// SIMATIC S7-200 project (STEP 7-Micro/WIN), CPU 222 REL 02.01

SYMBOL_TABLE USER1
AUTO             I0.0     // SELEZIONE MODO DI FUNZIONAMENTO AUTOMATICO
SEMI_AUTO        I0.1     // SELEZIONE MODO DI FUNZIONAMENTO SEMI-AUTOMATICO
MANU             I0.2     // SELEZIONE MODO DI FUNZIONAMENTO MANUALE
B7               I0.3     // TRASCINATORE
B8               I0.4     // TRASCINATORE
E1               I0.5     // ESPULSORE 1 MANUALE
E2               I0.6     // ESPULSORE 2 MANUALE
B1               I0.7     // RELE' FOTOELETTRICO
B2               I1.0     // RELE' FOTOELETTRICO
B3               I1.1     // RELE' FOTOELETTRICO
B4               I1.2     // RELE' FOTOELETTRICO BOX1
B5               I1.3     // RELE' FOTOELETTRICO BOX2
B6               I1.4     // RELE' FOTOELETTRICO FINE LINEA
MANU_RICH_TR     I1.5     // COMANDO MANUALE RICHIESTA TRONCHI
CORTO            M0.0     // RILEVATO TRONCO CORTO
MEDIO            M0.1     // RILEVATO TRONCO MEDIO
LUNGO            M0.2     // RILEVATO TRONCO LUNGO
MEM_T_EVAQ       M1.0     // MEMORIA PER CONSENTIRE L'USCITA DEL TRONCO A FINE LINEA
MEM_T_DEP_BOX2   M1.1     // MEMORIA MEMORIA PER CONSENTIRE IL DEPOSITO DEL TRONCO NEL BOX 2
MEM_T_DEP_BOX1   M1.2     // MEMORIA MEMORIA PER CONSENTIRE IL DEPOSITO DEL TRONCO NEL BOX 1
ESP1             Q0.0     // MOVIMENTO ESPULSORE 1
ESP2             Q0.1     // MOVIMENTO ESPULSORE 2
AUT_RICH_TR      Q0.2     // RICHIESTA TRONCHI
T_ATT_FINE       T39      // TEMPO ATTESA USCTA SU FINE LINEA
T_ATT_BOX_2      T40      // TEMPO ATTESA DEPOSITO SU BOX 2
T_ATT_BOX_1      T41      // TEMPO ATTESA DEPOSITO SU BOX  1
END_SYMBOL_TABLE

ORGANIZATION_BLOCK MAIN:OB1
TITLE=DP208 SELEZIONE LUNGHEZZE
BEGIN
Network 1 // COMMUTA SUL FUNZIONAMENTO MANUALE
LD     MANU:I0.2
CALL   MANUALE:SBR3
Network 2 // COMMUTA SUL FUNZIONAMENTO SEMI AUTOMATICO
LD     SEMI_AUTO:I0.1
CALL   SEMIAUTOMATICO:SBR0
Network 3 // COMMUTA SUL FUNZIONAMENTO AUTOMATICO
LD     AUTO:I0.0
CALL   AUTOMATICO:SBR1
Network 4 // ESEGUE LA SELEZIONE DEL FORMATO 
LD     SM0.0
CALL   SELEZIONE:SBR2
END_ORGANIZATION_BLOCK

SUBROUTINE_BLOCK SEMIAUTOMATICO:SBR0
TITLE=FUNZIONAMENTO SEMI-AUTOMATICO
BEGIN
Network 1 // RICHIAMO TRONCO
// RICHIAMO TRONCHI:
// - RICHIESTA MANUALE DA PULSANTE
// - RICHIESTA AUTOMATICA DOPO ATTESA TRANSITO COMPLETO DEL TRONCO PRECEDENTE
LD     T_ATT_FINE:T39
O      T_ATT_BOX_2:T40
O      T_ATT_BOX_1:T41
O      MANU_RICH_TR:I1.5
=      AUT_RICH_TR:Q0.2
=      Q0.3
Network 2 // USCITA TRONCO LUNGO
// RITARDO INTENZIONALE PRIMA DI RICHIAMARE IL TRONCO SUCCESSIVO
// PER CONSENTIRE L'USCITA DEL TRONCO LUNGO
LD     B6:I1.4
ED
O      MEM_T_EVAQ:M1.0
LPS
AW<=   T_ATT_FINE:T39, 60
=      MEM_T_EVAQ:M1.0
LPP
TON    T_ATT_FINE:T39, +50
Network 3 // USCITA  TRONCO MEDIO
// RITARDO INTENZIONALE PRIMA DI RICHIAMARE IL TRONCO SUCCESSIVO
// PER CONSENTIRE IL DEPOSITO DEL TRONCO MEDIO NEL BOX 2
LD     B5:I1.3
ED
O      MEM_T_DEP_BOX2:M1.1
LPS
AW<=   T_ATT_BOX_2:T40, 30
=      MEM_T_DEP_BOX2:M1.1
LPP
TON    T_ATT_BOX_2:T40, 20
Network 4 // USCITA TRONCO CORTO
// RITARDO INTENZIONALE PRIMA DI RICHIAMARE IL TRONCO SUCCESSIVO
// PER CONSENTIRE IL DEPOSITO DEL TRONCO CORTO NEL BOX 1
LD     B4:I1.2
ED
O      MEM_T_DEP_BOX1:M1.2
LPS
AW<=   T_ATT_BOX_1:T41, 30
=      MEM_T_DEP_BOX1:M1.2
LPP
TON    T_ATT_BOX_1:T41, 20
Network 5 // COMANDO ESPULSORE 1
// SE IL TRONCO E' DEL FORMATO CORTO E VIENE COMANDATO L'ESPULSORE E1
// IL TRONCO VIENE DEPOSITATO NEL BOX 1
LD     CORTO:M0.0
A      E1:I0.5
=      ESP1:Q0.0
Network 6 // COMANDO ESPULSORE 2
// SE IL TRONCO E' DEL FORMATO MEDIO E VIENE COMANDATO L'ESPULSORE E2
// IL TRONCO VIENE DEPOSITATO NEL BOX 2
LD     MEDIO:M0.1
A      E2:I0.6
=      ESP2:Q0.1
Network 13 // Titolo del segmento
// Commento del segmento
END_SUBROUTINE_BLOCK

SUBROUTINE_BLOCK AUTOMATICO:SBR1
TITLE=FUNZIONAMENTO AUTOMATICO
BEGIN
Network 1 // RICHIAMO TRONCO
// RICHIAMO TRONCHI:
// - RICHIESTA MANUALE DA PULSANTE
// - RICHIESTA AUTOMATICA DOPO ATTESA TRANSITO COMPLETO DEL TRONCO PRECEDENTE
LD     T_ATT_FINE:T39
O      T_ATT_BOX_2:T40
O      T_ATT_BOX_1:T41
O      MANU_RICH_TR:I1.5
=      AUT_RICH_TR:Q0.2
=      Q0.3
Network 2 // USCITA TRONCO LUNGO
// RITARDO INTENZIONALE PRIMA DI RICHIAMARE IL TRONCO SUCCESSIVO
// PER CONSENTIRE L'USCITA DEL TRONCO LUNGO
LD     B6:I1.4
ED
O      MEM_T_EVAQ:M1.0
LPS
AW<=   T_ATT_FINE:T39, +60
=      MEM_T_EVAQ:M1.0
LPP
TON    T_ATT_FINE:T39, +50
Network 3 // DEPOSITO TRONCO MEDIO
// RITARDO INTENZIONALE PRIMA DI RICHIAMARE IL TRONCO SUCCESSIVO
// PER CONSENTIRE IL DEPOSITO DEL TRONCO MEDIO NEL BOX 2
LD     B5:I1.3
ED
O      MEM_T_DEP_BOX2:M1.1
LPS
AW<=   T_ATT_BOX_2:T40, 30
=      MEM_T_DEP_BOX2:M1.1
LPP
TON    T_ATT_BOX_2:T40, 20
Network 4 // DEPOSITO TRONCO CORTO
// RITARDO INTENZIONALE PRIMA DI RICHIAMARE IL TRONCO SUCCESSIVO
// PER CONSENTIRE IL DEPOSITO DEL TRONCO CORTO NEL BOX 1
LD     B4:I1.2
ED
O      MEM_T_DEP_BOX1:M1.2
LPS
AW<=   T_ATT_BOX_1:T41, 30
=      MEM_T_DEP_BOX1:M1.2
LPP
TON    T_ATT_BOX_1:T41, 20
Network 5 // COMANDO ESPULSORE 1
// AZIONAMENTO AUTOMATICO DELL'ESPULSORE 1:
// - E' STATO RILEVATO UN TRONCO CORTO
// - E' IMPEGNATO IL TRASCINATORE B7
LD     CORTO:M0.0
A      B7:I0.3
=      ESP1:Q0.0
Network 6 // COMANDO ESPULSORE 2
// AZIONAMENTO AUTOMATICO DELL'ESPULSORE 2:
// - E' STATO RILEVATO UN TRONCO MEDIO
// - E' IMPEGNATO IL TRASCINATORE B8
LD     MEDIO:M0.1
A      B8:I0.4
=      ESP2:Q0.1
END_SUBROUTINE_BLOCK

SUBROUTINE_BLOCK SELEZIONE:SBR2
TITLE=RICONOSCIMENTO FORMATO
BEGIN
Network 1 // RICONOSCIMENTO LUNGHEZZA
// RICONOSCE LA LUNGHEZZA IN BASE ALLA CONTEMPORANEITA' DELL'IMPEGNO DELLE FOTOCELLULE E
// MEMORIZZA IL FORMATO RILEVATO:
// - B1 TRONCO CORTO
// - B1+ B2 TRONCO MEDIO
// - B1 + B2 + B3 = TRONCO LUNGO
LD     SM0.0
LPS
A      B1:I0.7
EU
S      CORTO:M0.0, 1
R      MEDIO:M0.1, 2
LRD
A      B1:I0.7
A      B2:I1.0
EU
S      MEDIO:M0.1, 1
R      CORTO:M0.0, 1
R      LUNGO:M0.2, 1
LPP
A      B1:I0.7
A      B2:I1.0
A      B3:I1.1
EU
S      LUNGO:M0.2, 1
R      CORTO:M0.0, 2
Network 2 // Titolo del segmento
// Commento del segmento
END_SUBROUTINE_BLOCK

SUBROUTINE_BLOCK MANUALE:SBR3
TITLE=FUNZIONAMENTO  MANUALE
BEGIN
Network 1 // RICHIESTA TRONCO
// RICHIESTA TRONCO A DISCREZIONE DELL'OPERATORE MEDIANTE IL PULSANTE RICHIESTA TRONCHI
LD     MANU_RICH_TR:I1.5
O      Q0.3
AN     T_ATT_FINE:T39
=      AUT_RICH_TR:Q0.2
=      Q0.3
TON    T_ATT_FINE:T39, +15
Network 2 // AZIONAMENTO ESPULSORE 1
// AZIONAMENTO MANUALE DELL'ESPULSORE 1
// DEPOSITO NEL BOX 1 INDIPENDENTEMENTE DAL FORMATO A DISCREZIONE DELL'OPERATORE
LD     B3:I1.1
A      E1:I0.5
O      ESP1:Q0.0
AN     B7:I0.3
=      ESP1:Q0.0
Network 3 // AZIONAMENTO ESPULSORE 2
// AZIONAMENTO MANUALE DELL'ESPULSORE 2
// DEPOSITO NEL BOX 2 INDIPENDENTEMENTE DAL FORMATO A DISCREZIONE DELL'OPERATORE
LD     B3:I1.1
A      E2:I0.6
O      ESP2:Q0.1
AN     B8:I0.4
=      ESP2:Q0.1
Network 10 // Titolo del segmento
// Commento del segmento
Network 20 // Titolo del segmento
// Commento del segmento
END_SUBROUTINE_BLOCK
